FUNCTION_BLOCK FB_ManualControl
VAR_INPUT
	bEnable : BOOL;
	eMode : E_Mode;
	fJoyStickInput : REAL;
END_VAR
VAR_OUTPUT
	fManualControlOutput : LREAL;
END_VAR
VAR
	fbOpenLoopControl : FB_OpenLoopControl;

;END_VAR


IF bEnable = FALSE THEN
	RETURN;
END_IF

G_Parameter.fCylinderSpeedRef := G_Parameter.fMaxVelocity * G_Input.fJoyStickSignal;

fbOpenLoopControl
(
	bEnable := (G_Parameter.eMode = E_Mode.Manual),
	fVelocityReference_ms := G_Parameter.fCylinderSpeedRef,
	fMaxValveFlow_lmin := G_Parameter.fMaxVolumeFlow,
	fVelocityFeedForward => fManualControlOutput	
);

END_FUNCTION_BLOCK

(* stored: Version 1.1.0.1, ProductVersion 3.1.4024.10
   POU FB_ManualControl: Id {c3bab466-06a6-4c7e-b6e5-a4260602ff46}, SpecialFunc None *)
